// TIA Portal V21 export
DATA_BLOCK "Screensaver"   // DB37
{ S7_Optimized_Access := 'TRUE' }
// stored: MemoryReserve 100
   VAR
      Frameattuale : Int := 193;
      DecrementaFrame : Bool := FALSE;
      TipoScreenSaver : Int := 0;   // 0=compare,trasla,scompare 1=compare,trasla,scompare,compare,trasla,scompare 2=Compare,scompare 3=Compare,trasla,scompare,compare in mezzo,scompare in mezzo,trasla,scompare 4=Compare centrale, scompare centrale
      DurataFrame : "Std_stTimer";
   END_VAR
BEGIN
   DurataFrame.IN := TRUE;
   DurataFrame.O := FALSE;
   DurataFrame.Preset := 0.1;
   DurataFrame.TempoTrascorso := 0.1143518;
END_DATA_BLOCK
